// TIA Portal V18 export
// export: Created 2025-12-01T17:51:12.6725807Z, ExportSetting None, DisplayName Totally Integrated Automation Portal, DisplayVersion V18 Update 5, DisplayName TIA Portal Openness, DisplayVersion V18 Update 5, DisplayName TIA Portal Teamcenter Gateway, DisplayVersion V18, DisplayName TIA Portal Version Control Interface, DisplayVersion V18, DisplayName STEP 7 Professional, DisplayVersion V18 Update 5, DisplayName STEP 7 Safety, DisplayVersion V18, DisplayName WinCC Professional, DisplayVersion V18 Update 5
FUNCTION "KistlerPresser_Main" : Void   // FC2300, LAD
{ S7_Optimized_Access := 'TRUE' }
// stored: AutoNumber false, SetENOAutomatically false
   VAR_TEMP
      tRel : DInt;
   END_VAR
   VAR_TEMP   // added for the SCL form of the ladder/FBD networks
      _w1 : Bool;
   END_VAR
BEGIN

REGION Network 1: OP10_372A1 Kistler Press
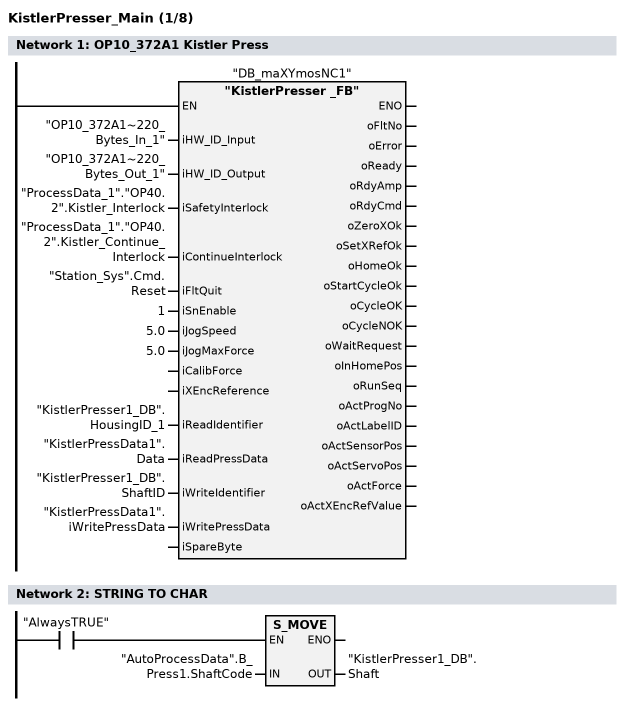
   RUNG wire#powerrail
      "DB_maXYmosNC1"(iHW_ID_Input := "OP10_372A1~220_Bytes_In_1", iHW_ID_Output := "OP10_372A1~220_Bytes_Out_1", iSafetyInterlock := "ProcessData_1"."OP40.2".Kistler_Interlock, iContinueInterlock := "ProcessData_1"."OP40.2".Kistler_Continue_Interlock, iFltQuit := "Station_Sys".Cmd.Reset, iSnEnable := 1, iJogSpeed := 5.0, iJogMaxForce := 5.0, iCalibForce :=, iXEncReference :=, iReadIdentifier := "KistlerPresser1_DB".HousingID_1, iReadPressData := "KistlerPressData1".Data, iWriteIdentifier := "KistlerPresser1_DB".ShaftID, iWritePressData := "KistlerPressData1".iWritePressData, iSpareByte :=, oFltNo =>, oError =>, oReady =>, oRdyAmp =>, oRdyCmd =>, oZeroXOk =>, oSetXRefOk =>, oHomeOk =>, oStartCycleOk =>, oCycleOK =>, oCycleNOK =>, oWaitRequest =>, oInHomePos =>, oRunSeq =>, oActProgNo =>, oActLabelID =>, oActSensorPos =>, oActServoPos =>, oActForce =>, oActXEncRefValue =>)
   END_RUNG
   // the same network as SCL:
   "DB_maXYmosNC1"(iHW_ID_Input := "OP10_372A1~220_Bytes_In_1",   // "KistlerPresser _FB"
                   iHW_ID_Output := "OP10_372A1~220_Bytes_Out_1",
                   iSafetyInterlock := "ProcessData_1"."OP40.2".Kistler_Interlock,
                   iContinueInterlock := "ProcessData_1"."OP40.2".Kistler_Continue_Interlock,
                   iFltQuit := "Station_Sys".Cmd.Reset,
                   iSnEnable := 1,
                   iJogSpeed := 5.0,
                   iJogMaxForce := 5.0,
                   iReadIdentifier := "KistlerPresser1_DB".HousingID_1,
                   iReadPressData := "KistlerPressData1".Data,
                   iWriteIdentifier := "KistlerPresser1_DB".ShaftID,
                   iWritePressData := "KistlerPressData1".iWritePressData);
END_REGION

REGION Network 2: STRING TO CHAR
   RUNG wire#powerrail
      Contact( "AlwaysTRUE" )
      S_Move(in := "AutoProcessData".B_Press1.ShaftCode, out => "KistlerPresser1_DB".Shaft)
   END_RUNG
   // the same network as SCL:
   IF "AlwaysTRUE" THEN "KistlerPresser1_DB".Shaft := "AutoProcessData".B_Press1.ShaftCode; END_IF;
END_REGION

REGION Network 3 (SCL): STRING TO CHAR
   Strg_TO_Chars(Strg:="KistlerPresser1_DB".Shaft,
                 pChars:=0,
                 Cnt=>#tRel,
                 Chars:="KistlerPresser1_DB".ShaftID);
END_REGION

REGION Network 4: OP10_372A1 Kistler Press_Safety_Interlock
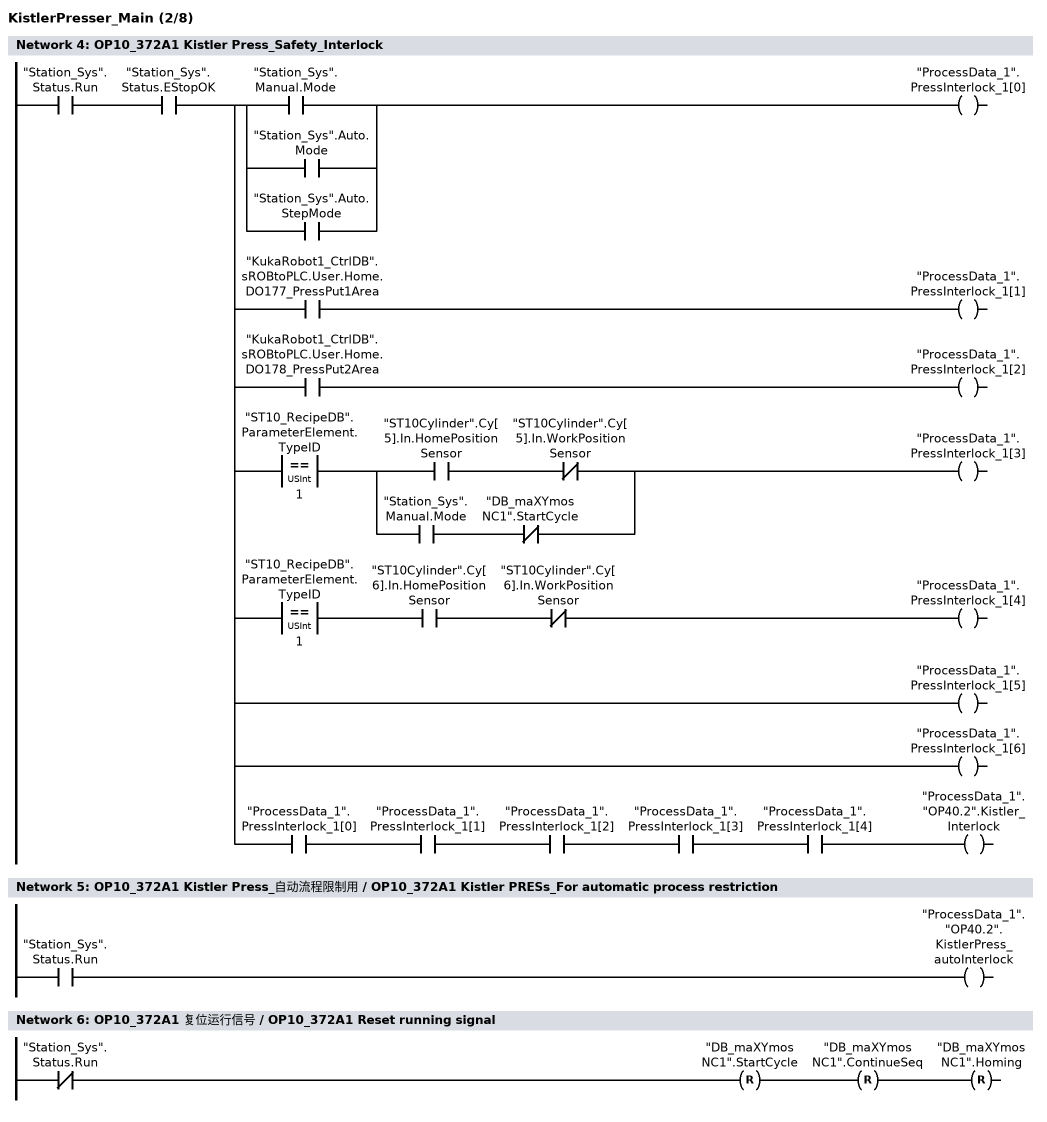
   RUNG wire#powerrail
      Contact( "Station_Sys".Status.Run )
      Contact( "Station_Sys".Status.EStopOK )
      wire#w1
      Contact( "Station_Sys".Manual.Mode )
      wire#w2
      Coil( "ProcessData_1".PressInterlock_1[0] )
   END_RUNG
   RUNG wire#w1
      Contact( "Station_Sys".Auto.Mode )
   END_RUNG wire#w2
   RUNG wire#w1
      Contact( "Station_Sys".Auto.StepMode )
   END_RUNG wire#w2
   RUNG wire#w1
      Contact( "KukaRobot1_CtrlDB".sROBtoPLC.User.Home.DO177_PressPut1Area )
      Coil( "ProcessData_1".PressInterlock_1[1] )
   END_RUNG
   RUNG wire#w1
      Contact( "KukaRobot1_CtrlDB".sROBtoPLC.User.Home.DO178_PressPut2Area )
      Coil( "ProcessData_1".PressInterlock_1[2] )
   END_RUNG
   RUNG wire#w1
      { S7_Templates := "SrcType := USInt" } EQ_Contact(in1 := "ST10_RecipeDB".ParameterElement.TypeID, in2 := 1)
      wire#w3
      Contact( "ST10Cylinder".Cy[5].In.HomePositionSensor )
      I_Contact( "ST10Cylinder".Cy[5].In.WorkPositionSensor )
      wire#w4
      Coil( "ProcessData_1".PressInterlock_1[3] )
   END_RUNG
   RUNG wire#w3
      Contact( "Station_Sys".Manual.Mode )
      I_Contact( "DB_maXYmosNC1".StartCycle )
   END_RUNG wire#w4
   RUNG wire#w1
      { S7_Templates := "SrcType := USInt" } EQ_Contact(in1 := "ST10_RecipeDB".ParameterElement.TypeID, in2 := 1)
      Contact( "ST10Cylinder".Cy[6].In.HomePositionSensor )
      I_Contact( "ST10Cylinder".Cy[6].In.WorkPositionSensor )
      Coil( "ProcessData_1".PressInterlock_1[4] )
   END_RUNG
   RUNG wire#w1
      Coil( "ProcessData_1".PressInterlock_1[5] )
   END_RUNG
   RUNG wire#w1
      Coil( "ProcessData_1".PressInterlock_1[6] )
   END_RUNG
   RUNG wire#w1
      Contact( "ProcessData_1".PressInterlock_1[0] )
      Contact( "ProcessData_1".PressInterlock_1[1] )
      Contact( "ProcessData_1".PressInterlock_1[2] )
      Contact( "ProcessData_1".PressInterlock_1[3] )
      Contact( "ProcessData_1".PressInterlock_1[4] )
      Coil( "ProcessData_1"."OP40.2".Kistler_Interlock )
   END_RUNG
   // the same network as SCL:
   #_w1 := "Station_Sys".Status.Run AND "Station_Sys".Status.EStopOK;
   "ProcessData_1".PressInterlock_1[0] := #_w1 AND ("Station_Sys".Manual.Mode OR "Station_Sys".Auto.Mode OR "Station_Sys".Auto.StepMode);
   "ProcessData_1".PressInterlock_1[1] := #_w1 AND "KukaRobot1_CtrlDB".sROBtoPLC.User.Home.DO177_PressPut1Area;
   "ProcessData_1".PressInterlock_1[2] := #_w1 AND "KukaRobot1_CtrlDB".sROBtoPLC.User.Home.DO178_PressPut2Area;
   "ProcessData_1".PressInterlock_1[3] := #_w1 AND ("ST10_RecipeDB".ParameterElement.TypeID = 1) AND (("ST10Cylinder".Cy[5].In.HomePositionSensor AND NOT "ST10Cylinder".Cy[5].In.WorkPositionSensor) OR ("Station_Sys".Manual.Mode AND NOT "DB_maXYmosNC1".StartCycle));
   "ProcessData_1".PressInterlock_1[4] := #_w1 AND ("ST10_RecipeDB".ParameterElement.TypeID = 1) AND "ST10Cylinder".Cy[6].In.HomePositionSensor AND NOT "ST10Cylinder".Cy[6].In.WorkPositionSensor;
   "ProcessData_1".PressInterlock_1[5] := #_w1;
   "ProcessData_1".PressInterlock_1[6] := #_w1;
   "ProcessData_1"."OP40.2".Kistler_Interlock := #_w1 AND "ProcessData_1".PressInterlock_1[0] AND "ProcessData_1".PressInterlock_1[1] AND "ProcessData_1".PressInterlock_1[2] AND "ProcessData_1".PressInterlock_1[3] AND "ProcessData_1".PressInterlock_1[4];
END_REGION

REGION Network 5: OP10_372A1 Kistler Press_自动流程限制用 / OP10_372A1 Kistler PRESs_For automatic process restriction
   RUNG wire#powerrail
      Contact( "Station_Sys".Status.Run )
      Coil( "ProcessData_1"."OP40.2".KistlerPress_autoInterlock )
   END_RUNG
   // the same network as SCL:
   "ProcessData_1"."OP40.2".KistlerPress_autoInterlock := "Station_Sys".Status.Run;
END_REGION

REGION Network 6: OP10_372A1 复位运行信号 / OP10_372A1 Reset running signal
   RUNG wire#powerrail
      I_Contact( "Station_Sys".Status.Run )
      R_Coil( "DB_maXYmosNC1".StartCycle )
      R_Coil( "DB_maXYmosNC1".ContinueSeq )
      R_Coil( "DB_maXYmosNC1".Homing )
   END_RUNG
   // the same network as SCL:
   IF NOT "Station_Sys".Status.Run THEN
       "DB_maXYmosNC1".StartCycle := FALSE;
       "DB_maXYmosNC1".ContinueSeq := FALSE;
       "DB_maXYmosNC1".Homing := FALSE;
   END_IF;
END_REGION

REGION Network 7: 手动模式程序号赋值 / Manual mode program number assignment
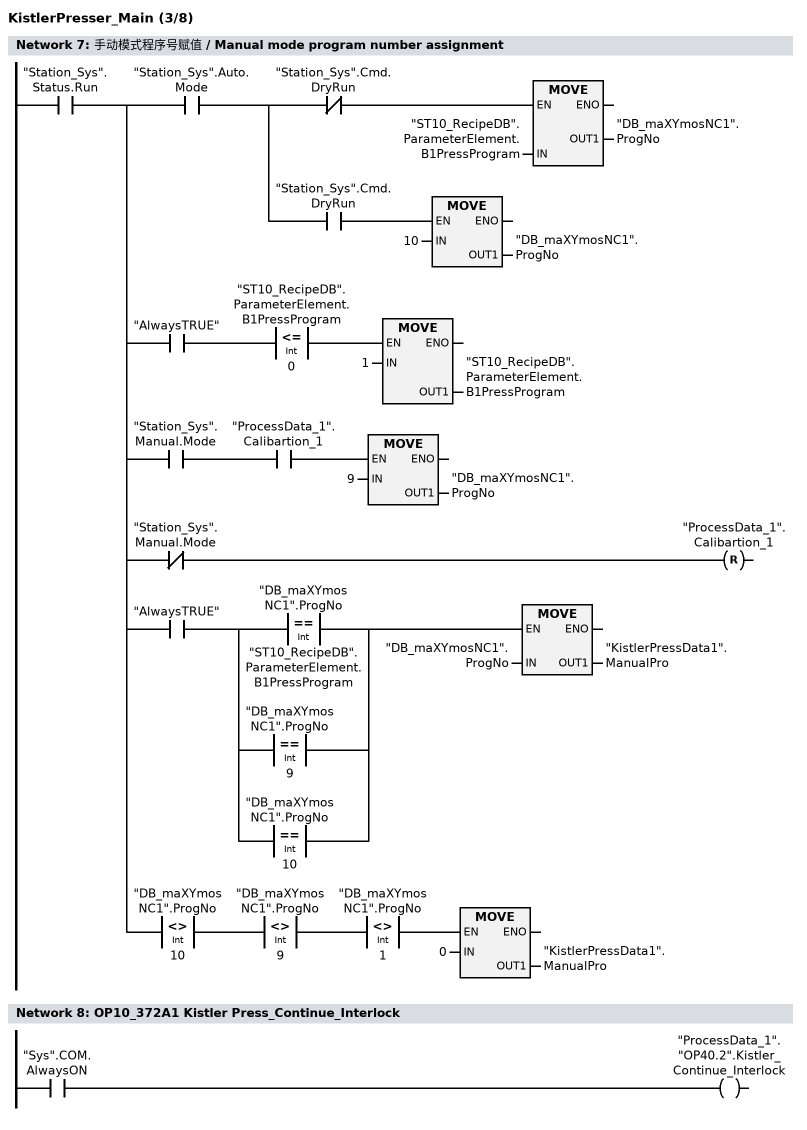
   RUNG wire#powerrail
      Contact( "Station_Sys".Status.Run )
      wire#w1
      Contact( "Station_Sys".Auto.Mode )
      wire#w2
      I_Contact( "Station_Sys".Cmd.DryRun )
      Move(in := "ST10_RecipeDB".ParameterElement.B1PressProgram, out1 => "DB_maXYmosNC1".ProgNo)
   END_RUNG
   RUNG wire#w2
      Contact( "Station_Sys".Cmd.DryRun )
      Move(in := 10, out1 => "DB_maXYmosNC1".ProgNo)
   END_RUNG
   RUNG wire#w1
      Contact( "AlwaysTRUE" )
      { S7_Templates := "SrcType := Int" } LE_Contact(in1 := "ST10_RecipeDB".ParameterElement.B1PressProgram, in2 := 0)
      Move(in := 1, out1 => "ST10_RecipeDB".ParameterElement.B1PressProgram)
   END_RUNG
   RUNG wire#w1
      Contact( "Station_Sys".Manual.Mode )
      Contact( "ProcessData_1".Calibartion_1 )
      Move(in := 9, out1 => "DB_maXYmosNC1".ProgNo)
   END_RUNG
   RUNG wire#w1
      I_Contact( "Station_Sys".Manual.Mode )
      R_Coil( "ProcessData_1".Calibartion_1 )
   END_RUNG
   RUNG wire#w1
      Contact( "AlwaysTRUE" )
      wire#w3
      { S7_Templates := "SrcType := Int" } EQ_Contact(in1 := "DB_maXYmosNC1".ProgNo, in2 := "ST10_RecipeDB".ParameterElement.B1PressProgram)
      wire#w4
      Move(in := "DB_maXYmosNC1".ProgNo, out1 => "KistlerPressData1".ManualPro)
   END_RUNG
   RUNG wire#w3
      { S7_Templates := "SrcType := Int" } EQ_Contact(in1 := "DB_maXYmosNC1".ProgNo, in2 := 9)
   END_RUNG wire#w4
   RUNG wire#w3
      { S7_Templates := "SrcType := Int" } EQ_Contact(in1 := "DB_maXYmosNC1".ProgNo, in2 := 10)
   END_RUNG wire#w4
   RUNG wire#w1
      { S7_Templates := "SrcType := Int" } NE_Contact(in1 := "DB_maXYmosNC1".ProgNo, in2 := 10)
      { S7_Templates := "SrcType := Int" } NE_Contact(in1 := "DB_maXYmosNC1".ProgNo, in2 := 9)
      { S7_Templates := "SrcType := Int" } NE_Contact(in1 := "DB_maXYmosNC1".ProgNo, in2 := 1)
      Move(in := 0, out1 => "KistlerPressData1".ManualPro)
   END_RUNG
   // the same network as SCL:
   #_w1 := "Station_Sys".Status.Run AND "Station_Sys".Auto.Mode;
   IF #_w1 AND NOT "Station_Sys".Cmd.DryRun THEN
       "DB_maXYmosNC1".ProgNo := "ST10_RecipeDB".ParameterElement.B1PressProgram;
   END_IF;
   IF #_w1 AND "Station_Sys".Cmd.DryRun THEN "DB_maXYmosNC1".ProgNo := 10; END_IF;
   IF "Station_Sys".Status.Run AND "AlwaysTRUE" AND ("ST10_RecipeDB".ParameterElement.B1PressProgram <= 0) THEN
       "ST10_RecipeDB".ParameterElement.B1PressProgram := 1;
   END_IF;
   IF "Station_Sys".Status.Run AND "Station_Sys".Manual.Mode AND "ProcessData_1".Calibartion_1 THEN
       "DB_maXYmosNC1".ProgNo := 9;
   END_IF;
   IF "Station_Sys".Status.Run AND NOT "Station_Sys".Manual.Mode THEN
       "ProcessData_1".Calibartion_1 := FALSE;
   END_IF;
   IF "Station_Sys".Status.Run AND "AlwaysTRUE" AND (("DB_maXYmosNC1".ProgNo = "ST10_RecipeDB".ParameterElement.B1PressProgram) OR ("DB_maXYmosNC1".ProgNo = 9) OR ("DB_maXYmosNC1".ProgNo = 10)) THEN
       "KistlerPressData1".ManualPro := "DB_maXYmosNC1".ProgNo;
   END_IF;
   IF "Station_Sys".Status.Run AND ("DB_maXYmosNC1".ProgNo <> 10) AND ("DB_maXYmosNC1".ProgNo <> 9) AND ("DB_maXYmosNC1".ProgNo <> 1) THEN
       "KistlerPressData1".ManualPro := 0;
   END_IF;
END_REGION

REGION Network 8: OP10_372A1 Kistler Press_Continue_Interlock
   RUNG wire#powerrail
      Contact( "Sys".COM.AlwaysON )
      Coil( "ProcessData_1"."OP40.2".Kistler_Continue_Interlock )
   END_RUNG
   // the same network as SCL:
   "ProcessData_1"."OP40.2".Kistler_Continue_Interlock := "Sys".COM.AlwaysON;
END_REGION

REGION Network 9: OP10_372A1 KistlerPressData 奇石乐第1次压装数据 / OP10_372A1 KistlerPressData The first KistlerPressdata
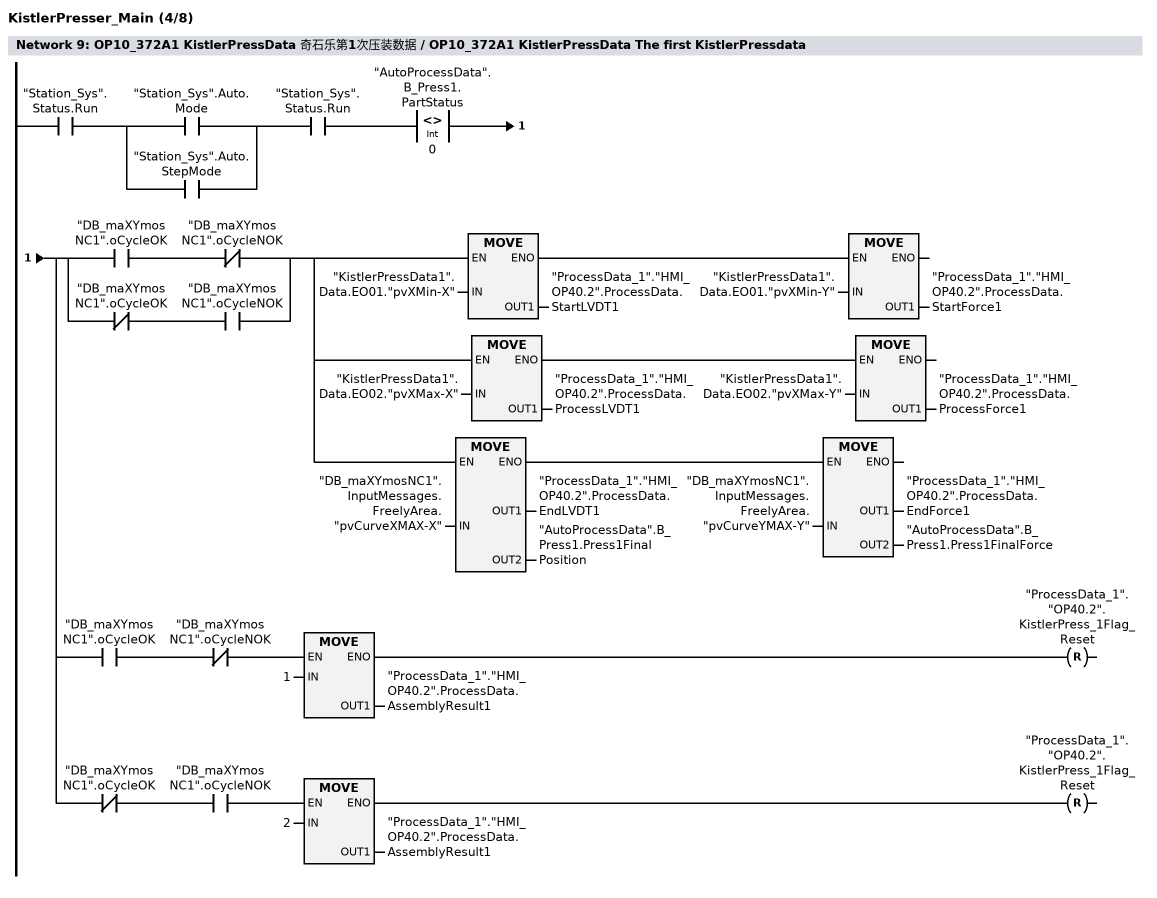
   RUNG wire#powerrail
      Contact( "Station_Sys".Status.Run )
      wire#w1
      Contact( "Station_Sys".Auto.Mode )
      wire#w2
      Contact( "Station_Sys".Status.Run )
      { S7_Templates := "SrcType := Int" } NE_Contact(in1 := "AutoProcessData".B_Press1.PartStatus, in2 := 0)
      wire#w3
      Contact( "DB_maXYmosNC1".oCycleOK )
      I_Contact( "DB_maXYmosNC1".oCycleNOK )
      wire#w4
      Move(in := "KistlerPressData1".Data.EO01."pvXMin-X", out1 => "ProcessData_1"."HMI_OP40.2".ProcessData.StartLVDT1)
      Move(in := "KistlerPressData1".Data.EO01."pvXMin-Y", out1 => "ProcessData_1"."HMI_OP40.2".ProcessData.StartForce1)
   END_RUNG
   RUNG wire#w1
      Contact( "Station_Sys".Auto.StepMode )
   END_RUNG wire#w2
   RUNG wire#w3
      I_Contact( "DB_maXYmosNC1".oCycleOK )
      Contact( "DB_maXYmosNC1".oCycleNOK )
   END_RUNG wire#w4
   RUNG wire#w4
      Move(in := "KistlerPressData1".Data.EO02."pvXMax-X", out1 => "ProcessData_1"."HMI_OP40.2".ProcessData.ProcessLVDT1)
      Move(in := "KistlerPressData1".Data.EO02."pvXMax-Y", out1 => "ProcessData_1"."HMI_OP40.2".ProcessData.ProcessForce1)
   END_RUNG
   RUNG wire#w4
      Move(in := "DB_maXYmosNC1".InputMessages.FreelyArea."pvCurveXMAX-X", out1 => "ProcessData_1"."HMI_OP40.2".ProcessData.EndLVDT1, out2 => "AutoProcessData".B_Press1.Press1FinalPosition)
      Move(in := "DB_maXYmosNC1".InputMessages.FreelyArea."pvCurveYMAX-Y", out1 => "ProcessData_1"."HMI_OP40.2".ProcessData.EndForce1, out2 => "AutoProcessData".B_Press1.Press1FinalForce)
   END_RUNG
   RUNG wire#w3
      Contact( "DB_maXYmosNC1".oCycleOK )
      I_Contact( "DB_maXYmosNC1".oCycleNOK )
      Move(in := 1, out1 => "ProcessData_1"."HMI_OP40.2".ProcessData.AssemblyResult1)
      R_Coil( "ProcessData_1"."OP40.2".KistlerPress_1Flag_Reset )
   END_RUNG
   RUNG wire#w3
      I_Contact( "DB_maXYmosNC1".oCycleOK )
      Contact( "DB_maXYmosNC1".oCycleNOK )
      Move(in := 2, out1 => "ProcessData_1"."HMI_OP40.2".ProcessData.AssemblyResult1)
      R_Coil( "ProcessData_1"."OP40.2".KistlerPress_1Flag_Reset )
   END_RUNG
   // the same network as SCL:
   #_w1 := "Station_Sys".Status.Run AND ("Station_Sys".Auto.Mode OR "Station_Sys".Auto.StepMode) AND "Station_Sys".Status.Run AND ("AutoProcessData".B_Press1.PartStatus <> 0);
   IF #_w1 AND (("DB_maXYmosNC1".oCycleOK AND NOT "DB_maXYmosNC1".oCycleNOK) OR (NOT "DB_maXYmosNC1".oCycleOK AND "DB_maXYmosNC1".oCycleNOK)) THEN
       "ProcessData_1"."HMI_OP40.2".ProcessData.StartLVDT1 := "KistlerPressData1".Data.EO01."pvXMin-X";
       "ProcessData_1"."HMI_OP40.2".ProcessData.StartForce1 := "KistlerPressData1".Data.EO01."pvXMin-Y";
       "ProcessData_1"."HMI_OP40.2".ProcessData.ProcessLVDT1 := "KistlerPressData1".Data.EO02."pvXMax-X";
       "ProcessData_1"."HMI_OP40.2".ProcessData.ProcessForce1 := "KistlerPressData1".Data.EO02."pvXMax-Y";
       "ProcessData_1"."HMI_OP40.2".ProcessData.EndLVDT1 := "DB_maXYmosNC1".InputMessages.FreelyArea."pvCurveXMAX-X";
       "AutoProcessData".B_Press1.Press1FinalPosition := "DB_maXYmosNC1".InputMessages.FreelyArea."pvCurveXMAX-X";
       "ProcessData_1"."HMI_OP40.2".ProcessData.EndForce1 := "DB_maXYmosNC1".InputMessages.FreelyArea."pvCurveYMAX-Y";
       "AutoProcessData".B_Press1.Press1FinalForce := "DB_maXYmosNC1".InputMessages.FreelyArea."pvCurveYMAX-Y";
   END_IF;
   IF #_w1 AND "DB_maXYmosNC1".oCycleOK AND NOT "DB_maXYmosNC1".oCycleNOK THEN
       "ProcessData_1"."HMI_OP40.2".ProcessData.AssemblyResult1 := 1;
       "ProcessData_1"."OP40.2".KistlerPress_1Flag_Reset := FALSE;
   END_IF;
   IF #_w1 AND NOT "DB_maXYmosNC1".oCycleOK AND "DB_maXYmosNC1".oCycleNOK THEN
       "ProcessData_1"."HMI_OP40.2".ProcessData.AssemblyResult1 := 2;
       "ProcessData_1"."OP40.2".KistlerPress_1Flag_Reset := FALSE;
   END_IF;
END_REGION

REGION Network 11: OP10_375A1 Kistler Press
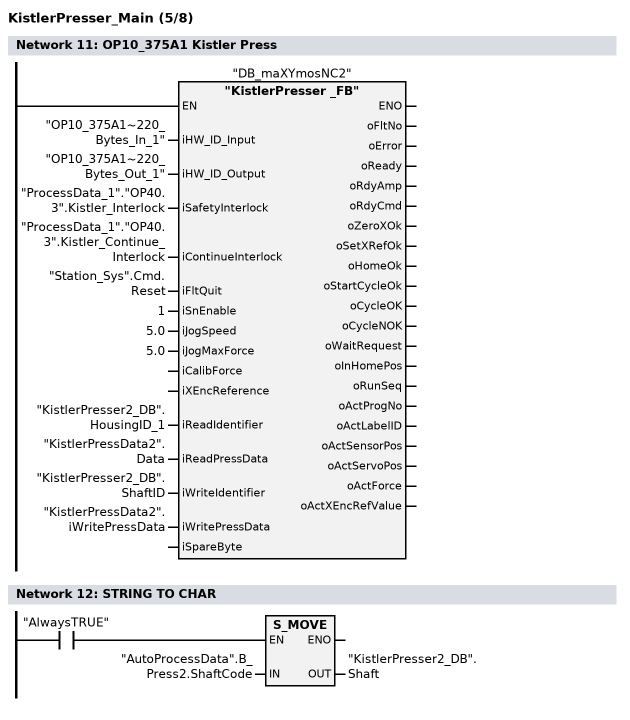
   RUNG wire#powerrail
      "DB_maXYmosNC2"(iHW_ID_Input := "OP10_375A1~220_Bytes_In_1", iHW_ID_Output := "OP10_375A1~220_Bytes_Out_1", iSafetyInterlock := "ProcessData_1"."OP40.3".Kistler_Interlock, iContinueInterlock := "ProcessData_1"."OP40.3".Kistler_Continue_Interlock, iFltQuit := "Station_Sys".Cmd.Reset, iSnEnable := 1, iJogSpeed := 5.0, iJogMaxForce := 5.0, iCalibForce :=, iXEncReference :=, iReadIdentifier := "KistlerPresser2_DB".HousingID_1, iReadPressData := "KistlerPressData2".Data, iWriteIdentifier := "KistlerPresser2_DB".ShaftID, iWritePressData := "KistlerPressData2".iWritePressData, iSpareByte :=, oFltNo =>, oError =>, oReady =>, oRdyAmp =>, oRdyCmd =>, oZeroXOk =>, oSetXRefOk =>, oHomeOk =>, oStartCycleOk =>, oCycleOK =>, oCycleNOK =>, oWaitRequest =>, oInHomePos =>, oRunSeq =>, oActProgNo =>, oActLabelID =>, oActSensorPos =>, oActServoPos =>, oActForce =>, oActXEncRefValue =>)
   END_RUNG
   // the same network as SCL:
   "DB_maXYmosNC2"(iHW_ID_Input := "OP10_375A1~220_Bytes_In_1",   // "KistlerPresser _FB"
                   iHW_ID_Output := "OP10_375A1~220_Bytes_Out_1",
                   iSafetyInterlock := "ProcessData_1"."OP40.3".Kistler_Interlock,
                   iContinueInterlock := "ProcessData_1"."OP40.3".Kistler_Continue_Interlock,
                   iFltQuit := "Station_Sys".Cmd.Reset,
                   iSnEnable := 1,
                   iJogSpeed := 5.0,
                   iJogMaxForce := 5.0,
                   iReadIdentifier := "KistlerPresser2_DB".HousingID_1,
                   iReadPressData := "KistlerPressData2".Data,
                   iWriteIdentifier := "KistlerPresser2_DB".ShaftID,
                   iWritePressData := "KistlerPressData2".iWritePressData);
END_REGION

REGION Network 12: STRING TO CHAR
   RUNG wire#powerrail
      Contact( "AlwaysTRUE" )
      S_Move(in := "AutoProcessData".B_Press2.ShaftCode, out => "KistlerPresser2_DB".Shaft)
   END_RUNG
   // the same network as SCL:
   IF "AlwaysTRUE" THEN "KistlerPresser2_DB".Shaft := "AutoProcessData".B_Press2.ShaftCode; END_IF;
END_REGION

REGION Network 13 (SCL): STRING TO CHAR
   Strg_TO_Chars(Strg:="KistlerPresser2_DB".Shaft,
                 pChars:=0,
                 Cnt=>#tRel,
                 Chars:="KistlerPresser2_DB".ShaftID);
END_REGION

REGION Network 14: OP10_375A1 Kistler Press_Safety_Interlock
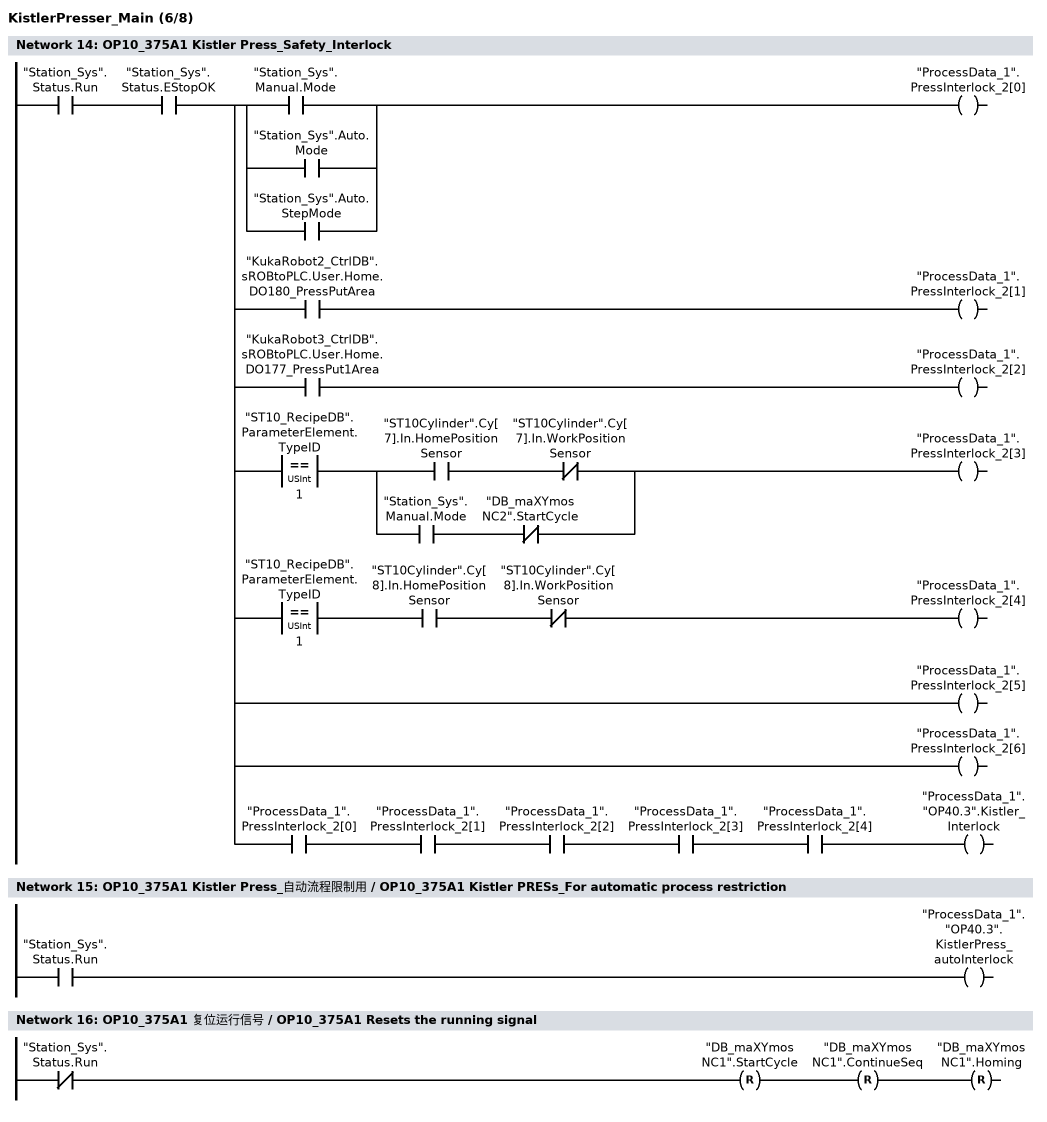
   RUNG wire#powerrail
      Contact( "Station_Sys".Status.Run )
      Contact( "Station_Sys".Status.EStopOK )
      wire#w1
      Contact( "Station_Sys".Manual.Mode )
      wire#w2
      Coil( "ProcessData_1".PressInterlock_2[0] )
   END_RUNG
   RUNG wire#w1
      Contact( "Station_Sys".Auto.Mode )
   END_RUNG wire#w2
   RUNG wire#w1
      Contact( "Station_Sys".Auto.StepMode )
   END_RUNG wire#w2
   RUNG wire#w1
      Contact( "KukaRobot2_CtrlDB".sROBtoPLC.User.Home.DO180_PressPutArea )
      Coil( "ProcessData_1".PressInterlock_2[1] )
   END_RUNG
   RUNG wire#w1
      Contact( "KukaRobot3_CtrlDB".sROBtoPLC.User.Home.DO177_PressPut1Area )
      Coil( "ProcessData_1".PressInterlock_2[2] )
   END_RUNG
   RUNG wire#w1
      { S7_Templates := "SrcType := USInt" } EQ_Contact(in1 := "ST10_RecipeDB".ParameterElement.TypeID, in2 := 1)
      wire#w3
      Contact( "ST10Cylinder".Cy[7].In.HomePositionSensor )
      I_Contact( "ST10Cylinder".Cy[7].In.WorkPositionSensor )
      wire#w4
      Coil( "ProcessData_1".PressInterlock_2[3] )
   END_RUNG
   RUNG wire#w3
      Contact( "Station_Sys".Manual.Mode )
      I_Contact( "DB_maXYmosNC2".StartCycle )
   END_RUNG wire#w4
   RUNG wire#w1
      { S7_Templates := "SrcType := USInt" } EQ_Contact(in1 := "ST10_RecipeDB".ParameterElement.TypeID, in2 := 1)
      Contact( "ST10Cylinder".Cy[8].In.HomePositionSensor )
      I_Contact( "ST10Cylinder".Cy[8].In.WorkPositionSensor )
      Coil( "ProcessData_1".PressInterlock_2[4] )
   END_RUNG
   RUNG wire#w1
      Coil( "ProcessData_1".PressInterlock_2[5] )
   END_RUNG
   RUNG wire#w1
      Coil( "ProcessData_1".PressInterlock_2[6] )
   END_RUNG
   RUNG wire#w1
      Contact( "ProcessData_1".PressInterlock_2[0] )
      Contact( "ProcessData_1".PressInterlock_2[1] )
      Contact( "ProcessData_1".PressInterlock_2[2] )
      Contact( "ProcessData_1".PressInterlock_2[3] )
      Contact( "ProcessData_1".PressInterlock_2[4] )
      Coil( "ProcessData_1"."OP40.3".Kistler_Interlock )
   END_RUNG
   // the same network as SCL:
   #_w1 := "Station_Sys".Status.Run AND "Station_Sys".Status.EStopOK;
   "ProcessData_1".PressInterlock_2[0] := #_w1 AND ("Station_Sys".Manual.Mode OR "Station_Sys".Auto.Mode OR "Station_Sys".Auto.StepMode);
   "ProcessData_1".PressInterlock_2[1] := #_w1 AND "KukaRobot2_CtrlDB".sROBtoPLC.User.Home.DO180_PressPutArea;
   "ProcessData_1".PressInterlock_2[2] := #_w1 AND "KukaRobot3_CtrlDB".sROBtoPLC.User.Home.DO177_PressPut1Area;
   "ProcessData_1".PressInterlock_2[3] := #_w1 AND ("ST10_RecipeDB".ParameterElement.TypeID = 1) AND (("ST10Cylinder".Cy[7].In.HomePositionSensor AND NOT "ST10Cylinder".Cy[7].In.WorkPositionSensor) OR ("Station_Sys".Manual.Mode AND NOT "DB_maXYmosNC2".StartCycle));
   "ProcessData_1".PressInterlock_2[4] := #_w1 AND ("ST10_RecipeDB".ParameterElement.TypeID = 1) AND "ST10Cylinder".Cy[8].In.HomePositionSensor AND NOT "ST10Cylinder".Cy[8].In.WorkPositionSensor;
   "ProcessData_1".PressInterlock_2[5] := #_w1;
   "ProcessData_1".PressInterlock_2[6] := #_w1;
   "ProcessData_1"."OP40.3".Kistler_Interlock := #_w1 AND "ProcessData_1".PressInterlock_2[0] AND "ProcessData_1".PressInterlock_2[1] AND "ProcessData_1".PressInterlock_2[2] AND "ProcessData_1".PressInterlock_2[3] AND "ProcessData_1".PressInterlock_2[4];
END_REGION

REGION Network 15: OP10_375A1 Kistler Press_自动流程限制用 / OP10_375A1 Kistler PRESs_For automatic process restriction
   RUNG wire#powerrail
      Contact( "Station_Sys".Status.Run )
      Coil( "ProcessData_1"."OP40.3".KistlerPress_autoInterlock )
   END_RUNG
   // the same network as SCL:
   "ProcessData_1"."OP40.3".KistlerPress_autoInterlock := "Station_Sys".Status.Run;
END_REGION

REGION Network 16: OP10_375A1 复位运行信号 / OP10_375A1 Resets the running signal
   RUNG wire#powerrail
      I_Contact( "Station_Sys".Status.Run )
      R_Coil( "DB_maXYmosNC1".StartCycle )
      R_Coil( "DB_maXYmosNC1".ContinueSeq )
      R_Coil( "DB_maXYmosNC1".Homing )
   END_RUNG
   // the same network as SCL:
   IF NOT "Station_Sys".Status.Run THEN
       "DB_maXYmosNC1".StartCycle := FALSE;
       "DB_maXYmosNC1".ContinueSeq := FALSE;
       "DB_maXYmosNC1".Homing := FALSE;
   END_IF;
END_REGION

REGION Network 17: 手动模式程序号赋值 / Manual mode program number assignment
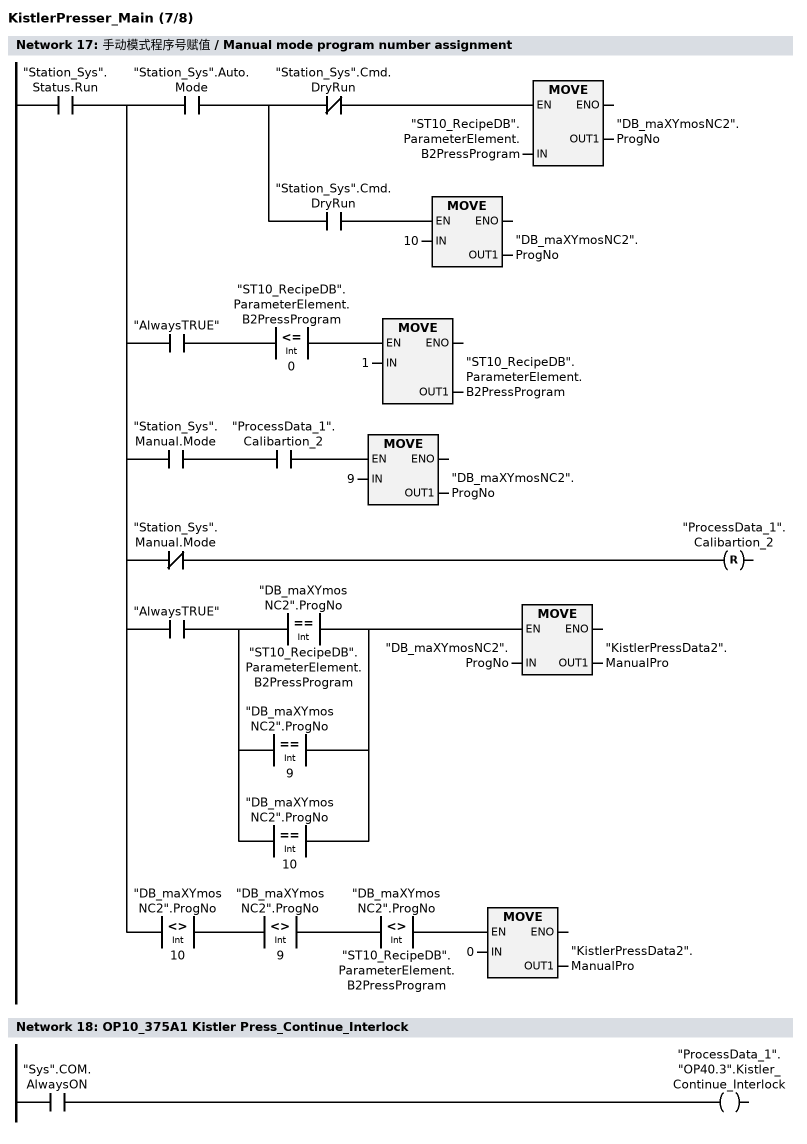
   RUNG wire#powerrail
      Contact( "Station_Sys".Status.Run )
      wire#w1
      Contact( "Station_Sys".Auto.Mode )
      wire#w2
      I_Contact( "Station_Sys".Cmd.DryRun )
      Move(in := "ST10_RecipeDB".ParameterElement.B2PressProgram, out1 => "DB_maXYmosNC2".ProgNo)
   END_RUNG
   RUNG wire#w2
      Contact( "Station_Sys".Cmd.DryRun )
      Move(in := 10, out1 => "DB_maXYmosNC2".ProgNo)
   END_RUNG
   RUNG wire#w1
      Contact( "AlwaysTRUE" )
      { S7_Templates := "SrcType := Int" } LE_Contact(in1 := "ST10_RecipeDB".ParameterElement.B2PressProgram, in2 := 0)
      Move(in := 1, out1 => "ST10_RecipeDB".ParameterElement.B2PressProgram)
   END_RUNG
   RUNG wire#w1
      Contact( "Station_Sys".Manual.Mode )
      Contact( "ProcessData_1".Calibartion_2 )
      Move(in := 9, out1 => "DB_maXYmosNC2".ProgNo)
   END_RUNG
   RUNG wire#w1
      I_Contact( "Station_Sys".Manual.Mode )
      R_Coil( "ProcessData_1".Calibartion_2 )
   END_RUNG
   RUNG wire#w1
      Contact( "AlwaysTRUE" )
      wire#w3
      { S7_Templates := "SrcType := Int" } EQ_Contact(in1 := "DB_maXYmosNC2".ProgNo, in2 := "ST10_RecipeDB".ParameterElement.B2PressProgram)
      wire#w4
      Move(in := "DB_maXYmosNC2".ProgNo, out1 => "KistlerPressData2".ManualPro)
   END_RUNG
   RUNG wire#w3
      { S7_Templates := "SrcType := Int" } EQ_Contact(in1 := "DB_maXYmosNC2".ProgNo, in2 := 9)
   END_RUNG wire#w4
   RUNG wire#w3
      { S7_Templates := "SrcType := Int" } EQ_Contact(in1 := "DB_maXYmosNC2".ProgNo, in2 := 10)
   END_RUNG wire#w4
   RUNG wire#w1
      { S7_Templates := "SrcType := Int" } NE_Contact(in1 := "DB_maXYmosNC2".ProgNo, in2 := 10)
      { S7_Templates := "SrcType := Int" } NE_Contact(in1 := "DB_maXYmosNC2".ProgNo, in2 := 9)
      { S7_Templates := "SrcType := Int" } NE_Contact(in1 := "DB_maXYmosNC2".ProgNo, in2 := "ST10_RecipeDB".ParameterElement.B2PressProgram)
      Move(in := 0, out1 => "KistlerPressData2".ManualPro)
   END_RUNG
   // the same network as SCL:
   #_w1 := "Station_Sys".Status.Run AND "Station_Sys".Auto.Mode;
   IF #_w1 AND NOT "Station_Sys".Cmd.DryRun THEN
       "DB_maXYmosNC2".ProgNo := "ST10_RecipeDB".ParameterElement.B2PressProgram;
   END_IF;
   IF #_w1 AND "Station_Sys".Cmd.DryRun THEN "DB_maXYmosNC2".ProgNo := 10; END_IF;
   IF "Station_Sys".Status.Run AND "AlwaysTRUE" AND ("ST10_RecipeDB".ParameterElement.B2PressProgram <= 0) THEN
       "ST10_RecipeDB".ParameterElement.B2PressProgram := 1;
   END_IF;
   IF "Station_Sys".Status.Run AND "Station_Sys".Manual.Mode AND "ProcessData_1".Calibartion_2 THEN
       "DB_maXYmosNC2".ProgNo := 9;
   END_IF;
   IF "Station_Sys".Status.Run AND NOT "Station_Sys".Manual.Mode THEN
       "ProcessData_1".Calibartion_2 := FALSE;
   END_IF;
   IF "Station_Sys".Status.Run AND "AlwaysTRUE" AND (("DB_maXYmosNC2".ProgNo = "ST10_RecipeDB".ParameterElement.B2PressProgram) OR ("DB_maXYmosNC2".ProgNo = 9) OR ("DB_maXYmosNC2".ProgNo = 10)) THEN
       "KistlerPressData2".ManualPro := "DB_maXYmosNC2".ProgNo;
   END_IF;
   IF "Station_Sys".Status.Run AND ("DB_maXYmosNC2".ProgNo <> 10) AND ("DB_maXYmosNC2".ProgNo <> 9) AND ("DB_maXYmosNC2".ProgNo <> "ST10_RecipeDB".ParameterElement.B2PressProgram) THEN
       "KistlerPressData2".ManualPro := 0;
   END_IF;
END_REGION

REGION Network 18: OP10_375A1 Kistler Press_Continue_Interlock
   RUNG wire#powerrail
      Contact( "Sys".COM.AlwaysON )
      Coil( "ProcessData_1"."OP40.3".Kistler_Continue_Interlock )
   END_RUNG
   // the same network as SCL:
   "ProcessData_1"."OP40.3".Kistler_Continue_Interlock := "Sys".COM.AlwaysON;
END_REGION

REGION Network 19: OP10_375A1 KistlerPressData 奇石乐第1次压装数据 / OP10_375A1 KistlerPressData The first KistlerPressdata
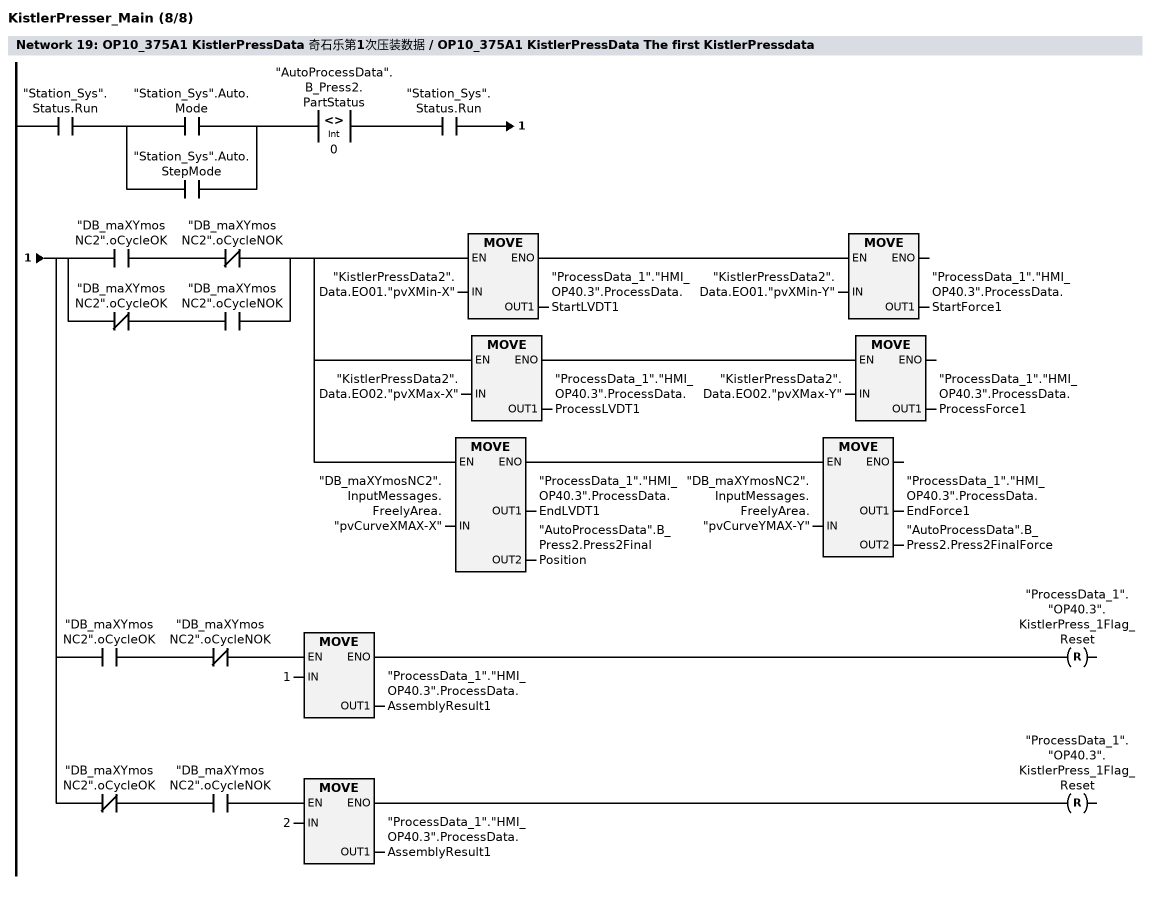
   RUNG wire#powerrail
      Contact( "Station_Sys".Status.Run )
      wire#w1
      Contact( "Station_Sys".Auto.Mode )
      wire#w2
      { S7_Templates := "SrcType := Int" } NE_Contact(in1 := "AutoProcessData".B_Press2.PartStatus, in2 := 0)
      Contact( "Station_Sys".Status.Run )
      wire#w3
      Contact( "DB_maXYmosNC2".oCycleOK )
      I_Contact( "DB_maXYmosNC2".oCycleNOK )
      wire#w4
      Move(in := "KistlerPressData2".Data.EO01."pvXMin-X", out1 => "ProcessData_1"."HMI_OP40.3".ProcessData.StartLVDT1)
      Move(in := "KistlerPressData2".Data.EO01."pvXMin-Y", out1 => "ProcessData_1"."HMI_OP40.3".ProcessData.StartForce1)
   END_RUNG
   RUNG wire#w1
      Contact( "Station_Sys".Auto.StepMode )
   END_RUNG wire#w2
   RUNG wire#w3
      I_Contact( "DB_maXYmosNC2".oCycleOK )
      Contact( "DB_maXYmosNC2".oCycleNOK )
   END_RUNG wire#w4
   RUNG wire#w4
      Move(in := "KistlerPressData2".Data.EO02."pvXMax-X", out1 => "ProcessData_1"."HMI_OP40.3".ProcessData.ProcessLVDT1)
      Move(in := "KistlerPressData2".Data.EO02."pvXMax-Y", out1 => "ProcessData_1"."HMI_OP40.3".ProcessData.ProcessForce1)
   END_RUNG
   RUNG wire#w4
      Move(in := "DB_maXYmosNC2".InputMessages.FreelyArea."pvCurveXMAX-X", out1 => "ProcessData_1"."HMI_OP40.3".ProcessData.EndLVDT1, out2 => "AutoProcessData".B_Press2.Press2FinalPosition)
      Move(in := "DB_maXYmosNC2".InputMessages.FreelyArea."pvCurveYMAX-Y", out1 => "ProcessData_1"."HMI_OP40.3".ProcessData.EndForce1, out2 => "AutoProcessData".B_Press2.Press2FinalForce)
   END_RUNG
   RUNG wire#w3
      Contact( "DB_maXYmosNC2".oCycleOK )
      I_Contact( "DB_maXYmosNC2".oCycleNOK )
      Move(in := 1, out1 => "ProcessData_1"."HMI_OP40.3".ProcessData.AssemblyResult1)
      R_Coil( "ProcessData_1"."OP40.3".KistlerPress_1Flag_Reset )
   END_RUNG
   RUNG wire#w3
      I_Contact( "DB_maXYmosNC2".oCycleOK )
      Contact( "DB_maXYmosNC2".oCycleNOK )
      Move(in := 2, out1 => "ProcessData_1"."HMI_OP40.3".ProcessData.AssemblyResult1)
      R_Coil( "ProcessData_1"."OP40.3".KistlerPress_1Flag_Reset )
   END_RUNG
   // the same network as SCL:
   #_w1 := "Station_Sys".Status.Run AND ("Station_Sys".Auto.Mode OR "Station_Sys".Auto.StepMode) AND ("AutoProcessData".B_Press2.PartStatus <> 0) AND "Station_Sys".Status.Run;
   IF #_w1 AND (("DB_maXYmosNC2".oCycleOK AND NOT "DB_maXYmosNC2".oCycleNOK) OR (NOT "DB_maXYmosNC2".oCycleOK AND "DB_maXYmosNC2".oCycleNOK)) THEN
       "ProcessData_1"."HMI_OP40.3".ProcessData.StartLVDT1 := "KistlerPressData2".Data.EO01."pvXMin-X";
       "ProcessData_1"."HMI_OP40.3".ProcessData.StartForce1 := "KistlerPressData2".Data.EO01."pvXMin-Y";
       "ProcessData_1"."HMI_OP40.3".ProcessData.ProcessLVDT1 := "KistlerPressData2".Data.EO02."pvXMax-X";
       "ProcessData_1"."HMI_OP40.3".ProcessData.ProcessForce1 := "KistlerPressData2".Data.EO02."pvXMax-Y";
       "ProcessData_1"."HMI_OP40.3".ProcessData.EndLVDT1 := "DB_maXYmosNC2".InputMessages.FreelyArea."pvCurveXMAX-X";
       "AutoProcessData".B_Press2.Press2FinalPosition := "DB_maXYmosNC2".InputMessages.FreelyArea."pvCurveXMAX-X";
       "ProcessData_1"."HMI_OP40.3".ProcessData.EndForce1 := "DB_maXYmosNC2".InputMessages.FreelyArea."pvCurveYMAX-Y";
       "AutoProcessData".B_Press2.Press2FinalForce := "DB_maXYmosNC2".InputMessages.FreelyArea."pvCurveYMAX-Y";
   END_IF;
   IF #_w1 AND "DB_maXYmosNC2".oCycleOK AND NOT "DB_maXYmosNC2".oCycleNOK THEN
       "ProcessData_1"."HMI_OP40.3".ProcessData.AssemblyResult1 := 1;
       "ProcessData_1"."OP40.3".KistlerPress_1Flag_Reset := FALSE;
   END_IF;
   IF #_w1 AND NOT "DB_maXYmosNC2".oCycleOK AND "DB_maXYmosNC2".oCycleNOK THEN
       "ProcessData_1"."HMI_OP40.3".ProcessData.AssemblyResult1 := 2;
       "ProcessData_1"."OP40.3".KistlerPress_1Flag_Reset := FALSE;
   END_IF;
END_REGION
END_FUNCTION
